(*---------------------------------------------------------------------------
 Copyright (c) 2018 BY mbc engineering GmbH, CH-6015 Luzern
 Licensed under the Apache License, Version 2.0
-----------------------------------------------------------------------------*)
// Command interface
INTERFACE ICommand

// The method is called in each cycle to execute the funktional part and the states of the command implementation.
METHOD Call
END_METHOD

END_INTERFACE

(* stored: Version 1.1.0.1, ProductVersion 3.1.4022.12
   Itf ICommand: Id {9dc6c476-c433-07d6-317f-3d274872f03c}
   Method Call: Id {b0863e7e-d159-0a36-1b9e-7efd24b9bd48} *)
